SUBAPPLICATION AuxInput_UP (* Subapplication Type *)
  (* Standard: 61499-2 *)
  (* Version 1.0, 2023-02-06, franz *)
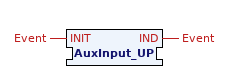
  EVENT_INPUT
    INIT;
  END_EVENT
  EVENT_OUTPUT
    IND;
  END_EVENT
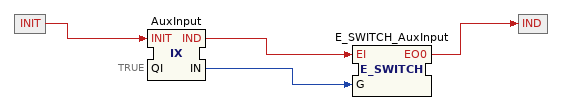
  FBS
    E_SWITCH_AuxInput : E_SWITCH;
    AuxInput : IX(QI := TRUE);
  END_FBS
  EVENT_CONNECTIONS
    AuxInput.IND TO E_SWITCH_AuxInput.EI;
    INIT TO AuxInput.INIT;
    E_SWITCH_AuxInput.EO0 TO IND;
  END_CONNECTIONS
  DATA_CONNECTIONS
    AuxInput.IN TO E_SWITCH_AuxInput.G;
  END_CONNECTIONS
END_SUBAPPLICATION
